(* Logix 5000 project; controller Project_Template vendor 1 type 14 code 106 rev 33.11; software revision 33.00 *)

TASK MainTask (continuous, watchdog 500 ms) : MainProgram

MODULES
   Local : vendor 1 type 14 code 106 (Compact 0, rev 33.11)
      Discrete_In_Slot_3 : 1769-IQ16 (Compact 3, rev 1.1, Input RPI 20 ms)
      Discrete_In_Slot_2 : 1769-IQ16 (Compact 2, rev 1.1, Input RPI 20 ms)
      ASCII_Slot_1 : vendor 1 type 109 code 66 (Compact 1, rev 2.1, Output RPI 2 ms)
      Discrete_Out_Slot_4 : 1769-OW16 (Compact 4, rev 1.1, Output RPI 20 ms)
      Discrete_Out_Slot_5 : 1769-OW16 (Compact 5, rev 1.1, Output RPI 20 ms)
END_MODULES

TYPE BCR_Data :
STRUCT
   LEN : DINT;
   DATA : SINT[9];
END_STRUCT
END_TYPE

TYPE Color_Data :
STRUCT
   LEN : DINT;
   DATA : SINT[4];
END_STRUCT
END_TYPE

VAR_GLOBAL   (* controller tags *)
   I_Auto_Mode_Selector : ALIAS FOR Local:2:I.Data.2;
   I_Barcode_Stop_Raised : ALIAS FOR Local:3:I.Data.1;
   I_Box_Ejector_Extended : ALIAS FOR Local:2:I.Data.4;
   I_Exit_Proxy : ALIAS FOR Local:3:I.Data.7;
   I_Reject_Cyl_Lowered : ALIAS FOR Local:3:I.Data.2;
   I_Reset_PB : ALIAS FOR Local:2:I.Data.3;
   I_Start_PB : ALIAS FOR Local:2:I.Data.0;
   I_Stop_PB : ALIAS FOR Local:2:I.Data.1;
   I_Vacuum_Head_at_Conveyor : ALIAS FOR Local:3:I.Data.0;
   I_Vacuum_Head_at_Magazine : ALIAS FOR Local:2:I.Data.15;
   I_Vacuum_Head_Extended : ALIAS FOR Local:2:I.Data.14;
   I_Vacuum_Head_Lowered : ALIAS FOR Local:2:I.Data.10;
   I_Vacuum_Head_Raised : ALIAS FOR Local:2:I.Data.9;
   I_Vacuum_Head_Retracted : ALIAS FOR Local:2:I.Data.13;
   I_Vacuum_Head_Rotated_CCW : ALIAS FOR Local:2:I.Data.11;
   I_Vacuum_Head_Rotated_CW : ALIAS FOR Local:2:I.Data.12;
   I_Vacuum_Sensor_On : ALIAS FOR Local:3:I.Data.8;
   O_Amber_Tower_Ind : ALIAS FOR Local:5:O.Data.9;
   O_Barcode_Stop_Raise : ALIAS FOR Local:4:O.Data.14;
   O_Box_Eject : ALIAS FOR Local:4:O.Data.0;
   O_Conveyor_On : ALIAS FOR Local:5:O.Data.5;
   O_Green_Tower_Ind : ALIAS FOR Local:5:O.Data.8;
   O_Red_Tower_Ind : ALIAS FOR Local:5:O.Data.10;
   O_Reject_Cyl_Extend : ALIAS FOR Local:5:O.Data.0;
   O_Reject_Cyl_Lower : ALIAS FOR Local:4:O.Data.15;
   O_Vacuum_Head_Extend : ALIAS FOR Local:4:O.Data.8;
   O_Vacuum_Head_Lower : ALIAS FOR Local:4:O.Data.5;
   O_Vacuum_Head_Rotate_CCW : ALIAS FOR Local:4:O.Data.7;
   O_Vacuum_Head_Rotate_CW : ALIAS FOR Local:4:O.Data.6;
   O_Vacuum_Head_to_Conveyor : ALIAS FOR Local:4:O.Data.9;
   O_Vacuum_Head_to_Magazine : ALIAS FOR Local:4:O.Data.10;
   O_Vacuum_Off : ALIAS FOR Local:5:O.Data.2;
   O_Vacuum_On : ALIAS FOR Local:5:O.Data.1;
END_VAR

PROGRAM MainProgram   (* main routine MainRoutine *)
VAR
   barcode_timer : TIMER := (PRE := 3000);
   barcode_timer_1 : TIMER := (PRE := 1500);
   BCR_Good_Read : BOOL;
   BCR_Value : BCR_Data := '33320717$0D';
   Color_Code : DINT := 4;
   Color_Value : Color_Data := '2';
   complete : BOOL;
   Fast_Flash_Off : TIMER := (PRE := 250, ACC := 181, EN := 1, TT := 1);
   Fast_Flash_On : TIMER := (PRE := 250, ACC := 250, EN := 1, DN := 1);
   Fast_Flasher : BOOL := 1;
   Machine_Home : BOOL;
   New_Rx_ID : SINT := 118;
   next_box : BOOL;
   Normal_Flash_Off : TIMER := (PRE := 500);
   Normal_Flash_On : TIMER := (PRE := 500, ACC := 431, EN := 1, TT := 1);
   Old_Rx_ID : SINT := 118;
   Prod_Delay_Timer : TIMER[10] := ([0].PRE := 250, [0].ACC := 250, [0].EN := 1, [0].DN := 1, [1].PRE := 250, [2].PRE := 250, [3].PRE := 250, [4].PRE := 250, [5].PRE := 250, [6].PRE := 250, [7].PRE := 500, [8].PRE := 500);
   Prod_Running : BOOL := 1;
   prod_step : DINT;
   prod_test_bit : DINT := -1;
   Regular_flasher : BOOL;
   Reset_Delay_Timer : TIMER[10] := ([0].PRE := 250, [0].ACC := 250, [0].EN := 1, [0].DN := 1, [1].PRE := 250, [1].ACC := 250, [1].EN := 1, [1].DN := 1, [2].PRE := 250, [2].ACC := 250, [2].EN := 1, [2].DN := 1, [3].PRE := 250, [4].PRE := 250, [4].ACC := 250, [4].EN := 1, [4].DN := 1, [5].PRE := 250, [5].ACC := 250, [5].EN := 1, [5].DN := 1, [6].PRE := 250, [7].PRE := 250);
   Reset_step : DINT := 12;
   Reset_Test_Bit : DINT := -1;
   Resetting : BOOL;
   Slow_Flash_Off : TIMER := (PRE := 1000);
   Slow_Flash_ON : TIMER := (PRE := 1000, ACC := 431, EN := 1, TT := 1);
   Slow_Flasher : BOOL;
   stop_bit : BOOL;
   stop_flag : BOOL := 1;
   stopping : BOOL;
   Test_Bit : DINT;
END_VAR
VAR_INPUT
   dfzsgd : DINT;
END_VAR

ROUTINE a_Reset_Routine   (* ladder *)
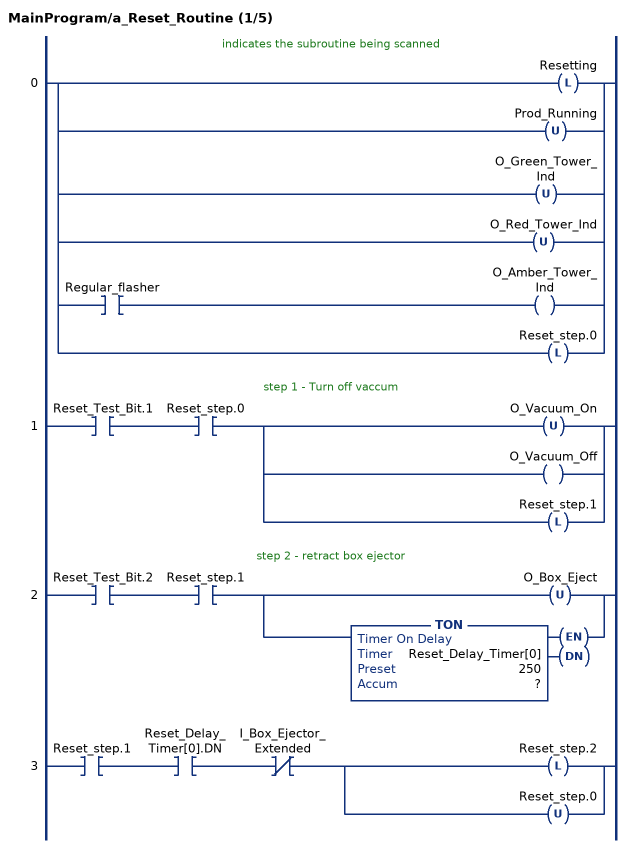
   // indicates the subroutine being scanned
   0: [OTL(Resetting) ,OTU(Prod_Running) ,OTU(O_Green_Tower_Ind) ,OTU(O_Red_Tower_Ind) ,XIC(Regular_flasher) OTE(O_Amber_Tower_Ind) ,OTL(Reset_step.0) ];
   // step 1 - Turn off vaccum
   1: XIC(Reset_Test_Bit.1)XIC(Reset_step.0)[OTU(O_Vacuum_On) ,OTE(O_Vacuum_Off) ,OTL(Reset_step.1) ];
   // step 2 - retract box ejector
   2: XIC(Reset_Test_Bit.2)XIC(Reset_step.1)[OTU(O_Box_Eject) ,TON(Reset_Delay_Timer[0],?,?) ];
   3: XIC(Reset_step.1)XIC(Reset_Delay_Timer[0].DN)XIO(I_Box_Ejector_Extended)[OTL(Reset_step.2) ,OTU(Reset_step.0) ];
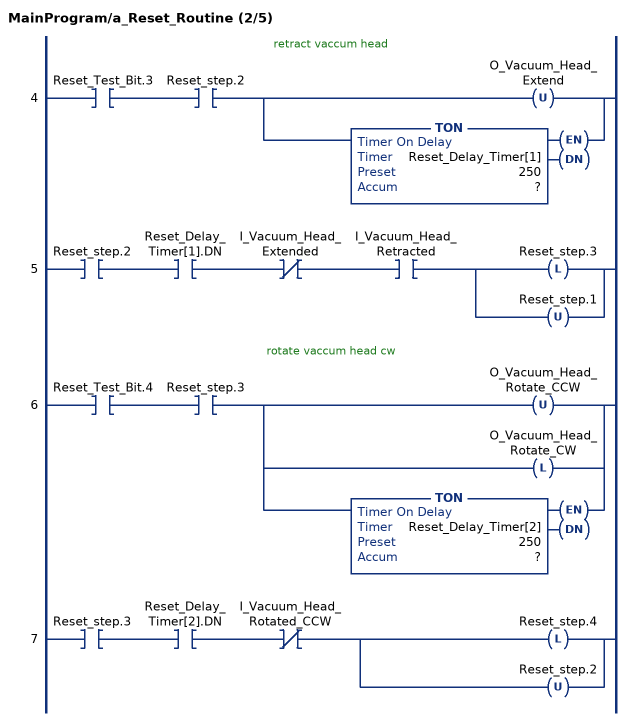
   // retract vaccum head
   4: XIC(Reset_Test_Bit.3)XIC(Reset_step.2)[OTU(O_Vacuum_Head_Extend) ,TON(Reset_Delay_Timer[1],?,?) ];
   5: XIC(Reset_step.2)XIC(Reset_Delay_Timer[1].DN)XIO(I_Vacuum_Head_Extended)XIC(I_Vacuum_Head_Retracted)[OTL(Reset_step.3) ,OTU(Reset_step.1) ];
   // rotate vaccum head cw
   6: XIC(Reset_Test_Bit.4)XIC(Reset_step.3)[OTU(O_Vacuum_Head_Rotate_CCW) ,OTL(O_Vacuum_Head_Rotate_CW) ,TON(Reset_Delay_Timer[2],?,?) ];
   7: XIC(Reset_step.3)XIC(Reset_Delay_Timer[2].DN)XIO(I_Vacuum_Head_Rotated_CCW)[OTL(Reset_step.4) ,OTU(Reset_step.2) ];
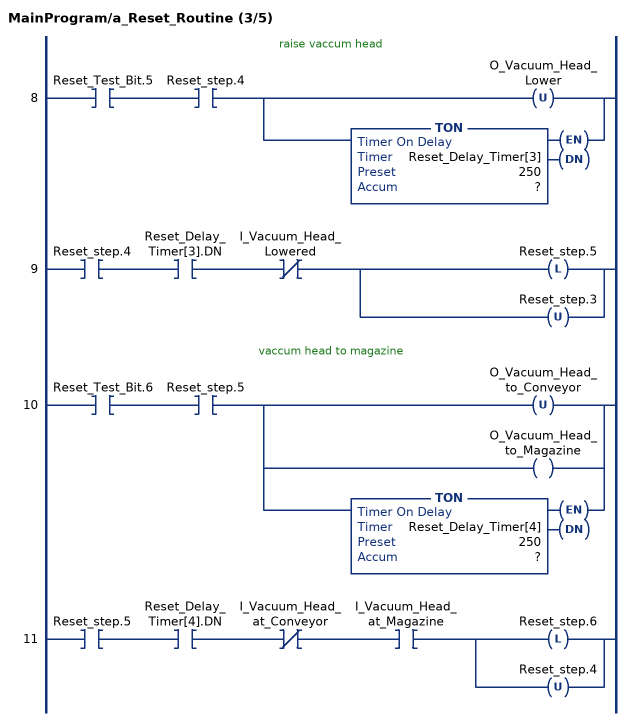
   // raise vaccum head
   8: XIC(Reset_Test_Bit.5)XIC(Reset_step.4)[OTU(O_Vacuum_Head_Lower) ,TON(Reset_Delay_Timer[3],?,?) ];
   9: XIC(Reset_step.4)XIC(Reset_Delay_Timer[3].DN)XIO(I_Vacuum_Head_Lowered)[OTL(Reset_step.5) ,OTU(Reset_step.3) ];
   // vaccum head to magazine
   10: XIC(Reset_Test_Bit.6)XIC(Reset_step.5)[OTU(O_Vacuum_Head_to_Conveyor) ,OTE(O_Vacuum_Head_to_Magazine) ,TON(Reset_Delay_Timer[4],?,?) ];
   11: XIC(Reset_step.5)XIC(Reset_Delay_Timer[4].DN)XIO(I_Vacuum_Head_at_Conveyor)XIC(I_Vacuum_Head_at_Magazine)[OTL(Reset_step.6) ,OTU(Reset_step.4) ];
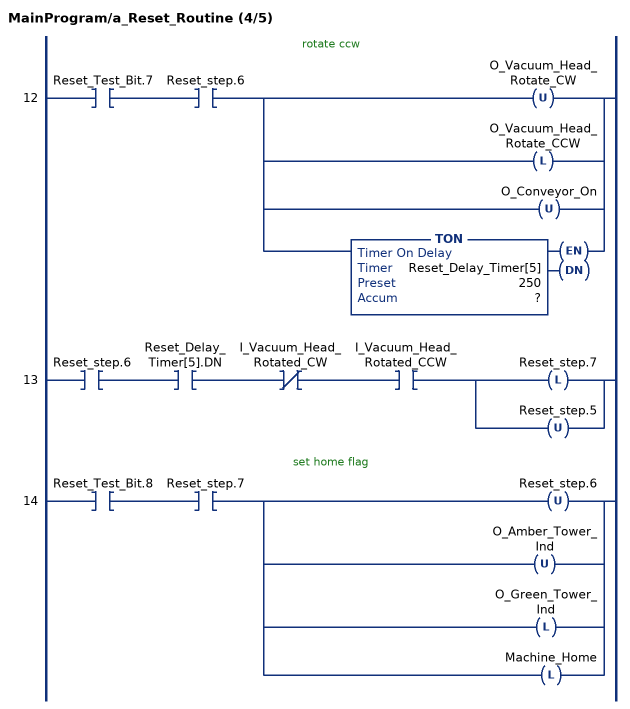
   // rotate ccw
   12: XIC(Reset_Test_Bit.7)XIC(Reset_step.6)[OTU(O_Vacuum_Head_Rotate_CW) ,OTL(O_Vacuum_Head_Rotate_CCW) ,OTU(O_Conveyor_On) ,TON(Reset_Delay_Timer[5],?,?) ];
   13: XIC(Reset_step.6)XIC(Reset_Delay_Timer[5].DN)XIO(I_Vacuum_Head_Rotated_CW)XIC(I_Vacuum_Head_Rotated_CCW)[OTL(Reset_step.7) ,OTU(Reset_step.5) ];
   // set home flag
   14: XIC(Reset_Test_Bit.8)XIC(Reset_step.7)[OTU(Reset_step.6) ,OTU(O_Amber_Tower_Ind) ,OTL(O_Green_Tower_Ind) ,OTL(Machine_Home) ];
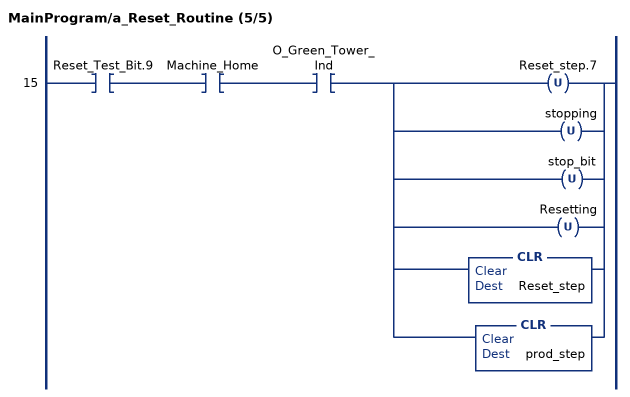
   15: XIC(Reset_Test_Bit.9)XIC(Machine_Home)XIC(O_Green_Tower_Ind)[OTU(Reset_step.7) ,OTU(stopping) ,OTU(stop_bit) ,OTU(Resetting) ,CLR(Reset_step) ,CLR(prod_step) ];
END_ROUTINE

ROUTINE Auto_Routine   (* ladder *)
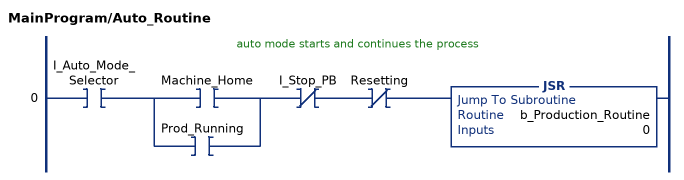
   // auto mode starts and continues the process
   0: XIC(I_Auto_Mode_Selector)[XIC(Machine_Home) ,XIC(Prod_Running) ]XIO(I_Stop_PB)XIO(Resetting)JSR(b_Production_Routine,0);
END_ROUTINE

ROUTINE b_Production_Routine   (* ladder *)
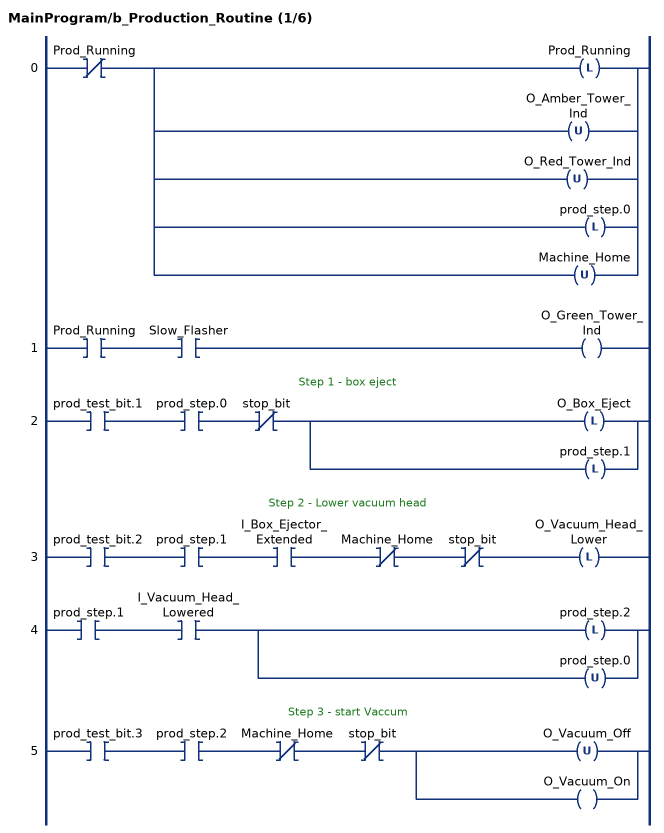
   0: XIO(Prod_Running)[OTL(Prod_Running) ,OTU(O_Amber_Tower_Ind) ,OTU(O_Red_Tower_Ind) ,OTL(prod_step.0) ,OTU(Machine_Home) ];
   1: XIC(Prod_Running)XIC(Slow_Flasher)OTE(O_Green_Tower_Ind);
   // Step 1 - box eject
   2: XIC(prod_test_bit.1)XIC(prod_step.0)XIO(stop_bit)[OTL(O_Box_Eject) ,OTL(prod_step.1) ];
   // Step 2 - Lower vacuum head
   3: XIC(prod_test_bit.2)XIC(prod_step.1)XIC(I_Box_Ejector_Extended)XIO(Machine_Home)XIO(stop_bit)OTL(O_Vacuum_Head_Lower);
   4: XIC(prod_step.1)XIC(I_Vacuum_Head_Lowered)[OTL(prod_step.2) ,OTU(prod_step.0) ];
   // Step 3 - start Vaccum
   5: XIC(prod_test_bit.3)XIC(prod_step.2)XIO(Machine_Home)XIO(stop_bit)[OTU(O_Vacuum_Off) ,OTE(O_Vacuum_On) ];
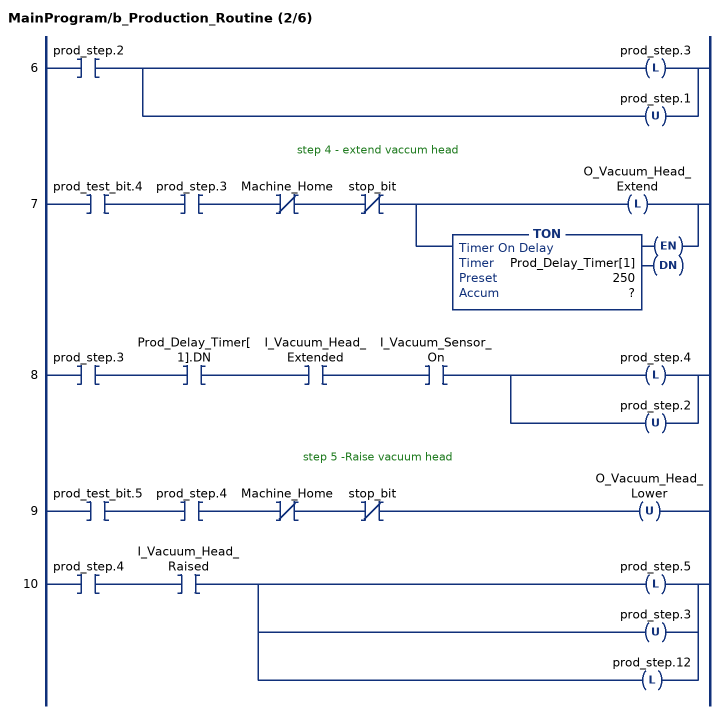
   6: XIC(prod_step.2)[OTL(prod_step.3) ,OTU(prod_step.1) ];
   // step 4 - extend vaccum head
   7: XIC(prod_test_bit.4)XIC(prod_step.3)XIO(Machine_Home)XIO(stop_bit)[OTL(O_Vacuum_Head_Extend) ,TON(Prod_Delay_Timer[1],?,?) ];
   8: XIC(prod_step.3)XIC(Prod_Delay_Timer[1].DN)XIC(I_Vacuum_Head_Extended)XIC(I_Vacuum_Sensor_On)[OTL(prod_step.4) ,OTU(prod_step.2) ];
   // step 5 -Raise vacuum head
   9: XIC(prod_test_bit.5)XIC(prod_step.4)XIO(Machine_Home)XIO(stop_bit)OTU(O_Vacuum_Head_Lower);
   10: XIC(prod_step.4)XIC(I_Vacuum_Head_Raised)[OTL(prod_step.5) ,OTU(prod_step.3) ,OTL(prod_step.12) ];
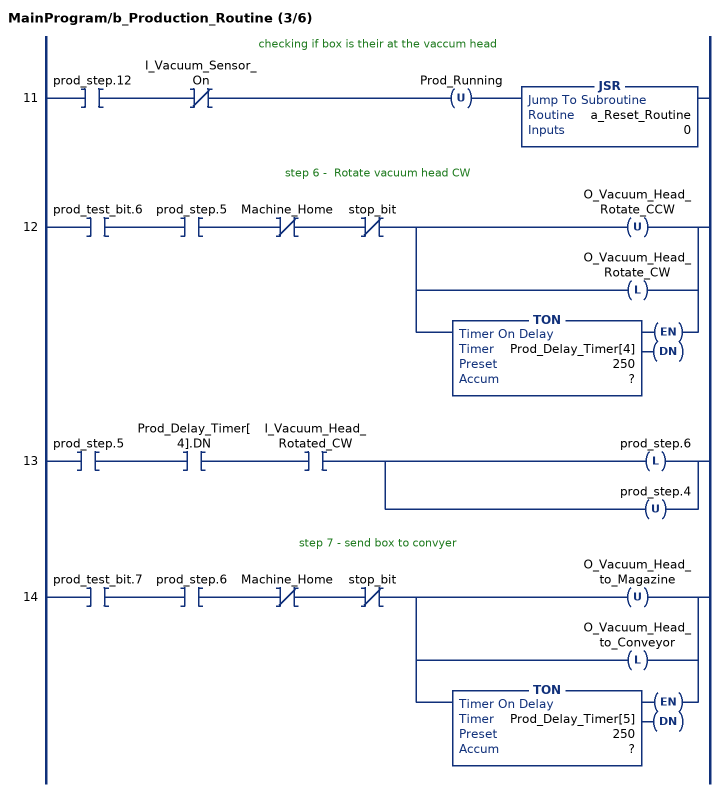
   // checking if box is their at the vaccum head
   11: XIC(prod_step.12)XIO(I_Vacuum_Sensor_On)OTU(Prod_Running)JSR(a_Reset_Routine,0);
   // step 6 -  Rotate vacuum head CW
   12: XIC(prod_test_bit.6)XIC(prod_step.5)XIO(Machine_Home)XIO(stop_bit)[OTU(O_Vacuum_Head_Rotate_CCW) ,OTL(O_Vacuum_Head_Rotate_CW) ,TON(Prod_Delay_Timer[4],?,?) ];
   13: XIC(prod_step.5)XIC(Prod_Delay_Timer[4].DN)XIC(I_Vacuum_Head_Rotated_CW)[OTL(prod_step.6) ,OTU(prod_step.4) ];
   // step 7 - send box to convyer
   14: XIC(prod_test_bit.7)XIC(prod_step.6)XIO(Machine_Home)XIO(stop_bit)[OTU(O_Vacuum_Head_to_Magazine) ,OTL(O_Vacuum_Head_to_Conveyor) ,TON(Prod_Delay_Timer[5],?,?) ];
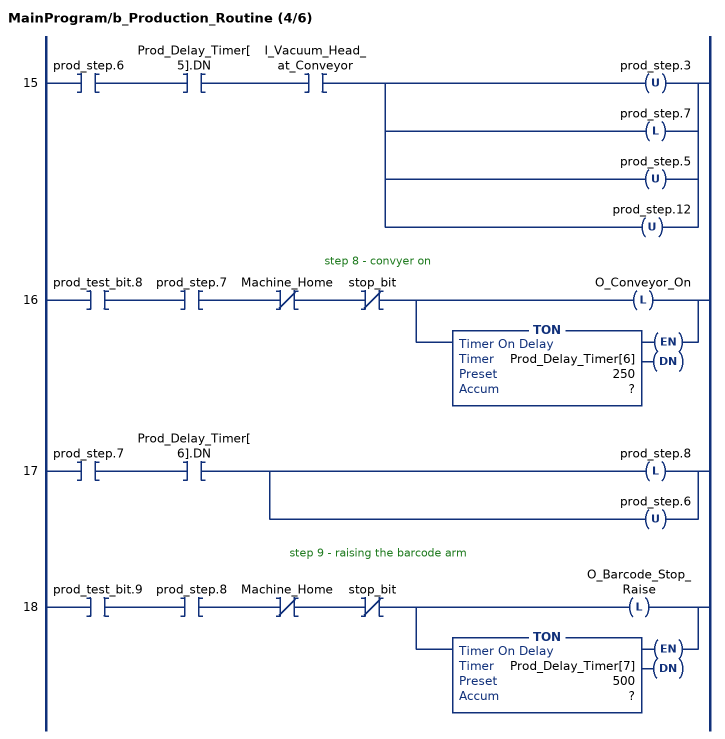
   15: XIC(prod_step.6)XIC(Prod_Delay_Timer[5].DN)XIC(I_Vacuum_Head_at_Conveyor)[OTU(prod_step.3) ,OTL(prod_step.7) ,OTU(prod_step.5) ,OTU(prod_step.12) ];
   // step 8 - convyer on
   16: XIC(prod_test_bit.8)XIC(prod_step.7)XIO(Machine_Home)XIO(stop_bit)[OTL(O_Conveyor_On) ,TON(Prod_Delay_Timer[6],?,?) ];
   17: XIC(prod_step.7)XIC(Prod_Delay_Timer[6].DN)[OTL(prod_step.8) ,OTU(prod_step.6) ];
   // step 9 - raising the barcode arm
   18: XIC(prod_test_bit.9)XIC(prod_step.8)XIO(Machine_Home)XIO(stop_bit)[OTL(O_Barcode_Stop_Raise) ,TON(Prod_Delay_Timer[7],?,?) ];
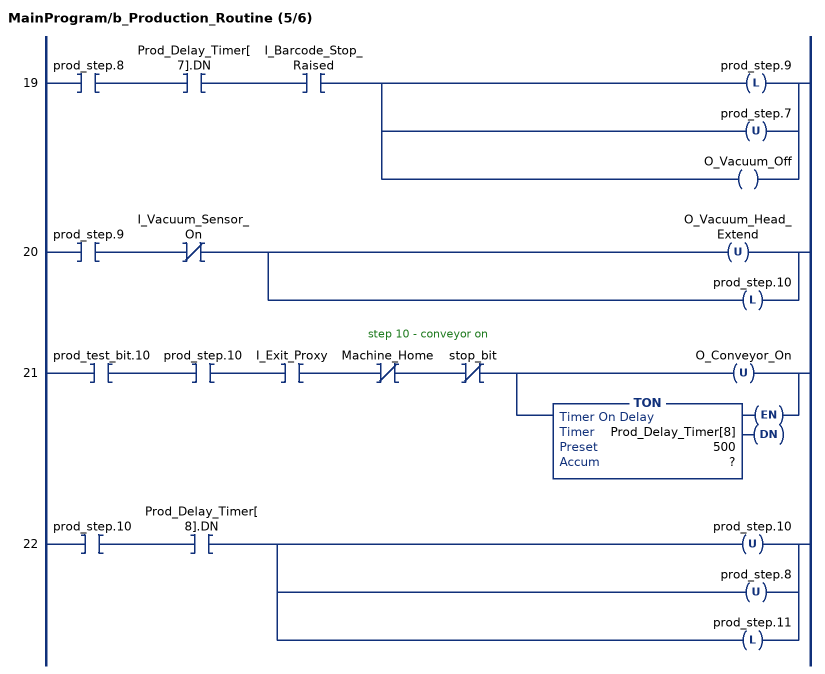
   19: XIC(prod_step.8)XIC(Prod_Delay_Timer[7].DN)XIC(I_Barcode_Stop_Raised)[OTL(prod_step.9) ,OTU(prod_step.7) ,OTE(O_Vacuum_Off) ];
   20: XIC(prod_step.9)XIO(I_Vacuum_Sensor_On)[OTU(O_Vacuum_Head_Extend) ,OTL(prod_step.10) ];
   // step 10 - conveyor on
   21: XIC(prod_test_bit.10)XIC(prod_step.10)XIC(I_Exit_Proxy)XIO(Machine_Home)XIO(stop_bit)[OTU(O_Conveyor_On) ,TON(Prod_Delay_Timer[8],?,?) ];
   22: XIC(prod_step.10)XIC(Prod_Delay_Timer[8].DN)[OTU(prod_step.10) ,OTU(prod_step.8) ,OTL(prod_step.11) ];
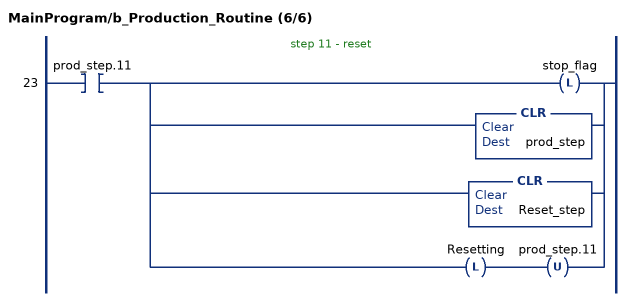
   // step 11 - reset
   23: XIC(prod_step.11)[OTL(stop_flag) ,CLR(prod_step) ,CLR(Reset_step) ,OTL(Resetting) OTU(prod_step.11) ];
END_ROUTINE

ROUTINE barcode_scan_routine   (* ladder *)
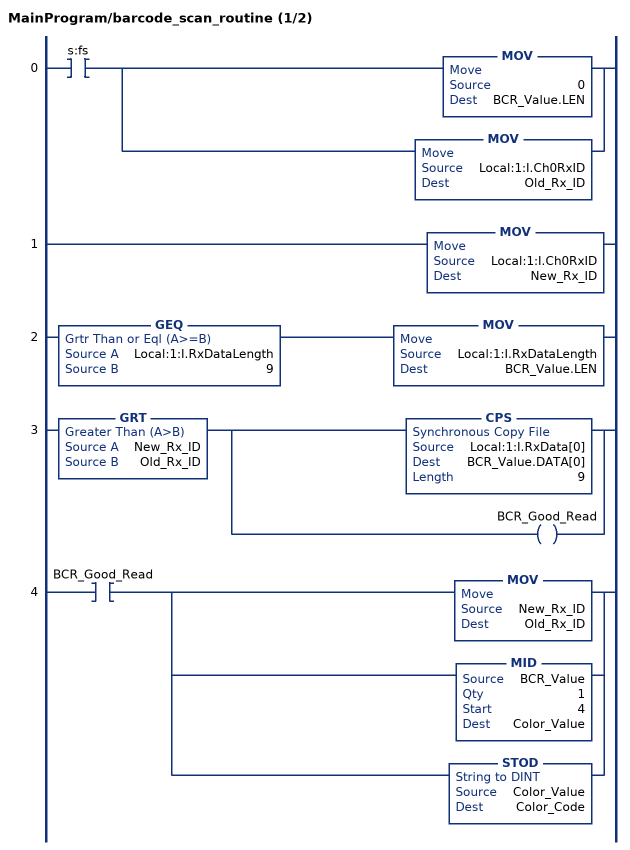
   0: XIC(s:fs)[MOV(0,BCR_Value.LEN) ,MOV(Local:1:I.Ch0RxID,Old_Rx_ID) ];
   1: MOV(Local:1:I.Ch0RxID,New_Rx_ID);
   2: GEQ(Local:1:I.RxDataLength,9)MOV(Local:1:I.RxDataLength,BCR_Value.LEN);
   3: GRT(New_Rx_ID,Old_Rx_ID)[CPS(Local:1:I.RxData[0],BCR_Value.DATA[0],9) ,OTE(BCR_Good_Read) ];
   4: XIC(BCR_Good_Read)[MOV(New_Rx_ID,Old_Rx_ID) ,MID(BCR_Value,1,4,Color_Value) ,STOD(Color_Value,Color_Code) ];
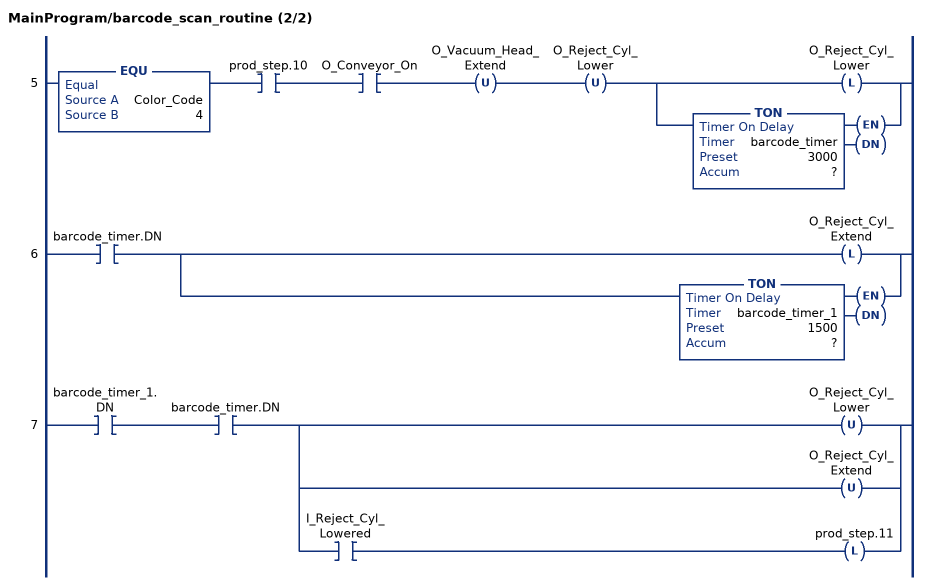
   5: EQU(Color_Code,4)XIC(prod_step.10)XIC(O_Conveyor_On)OTU(O_Vacuum_Head_Extend)OTU(O_Reject_Cyl_Lower)[OTL(O_Reject_Cyl_Lower) ,TON(barcode_timer,?,?) ];
   6: XIC(barcode_timer.DN)[OTL(O_Reject_Cyl_Extend) ,TON(barcode_timer_1,?,?) ];
   7: XIC(barcode_timer_1.DN)XIC(barcode_timer.DN)[OTU(O_Reject_Cyl_Lower) ,OTU(O_Reject_Cyl_Extend) ,XIC(I_Reject_Cyl_Lowered) OTL(prod_step.11) ];
END_ROUTINE

ROUTINE MainRoutine   (* ladder *)
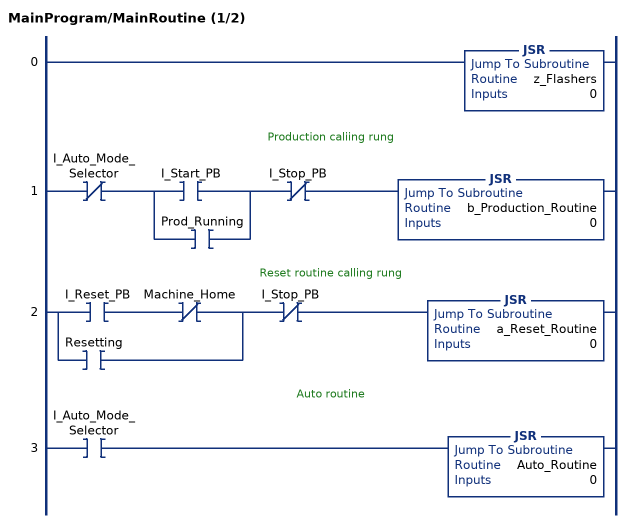
   0: JSR(z_Flashers,0);
   // Production caliing rung
   1: XIO(I_Auto_Mode_Selector)[XIC(I_Start_PB) ,XIC(Prod_Running) ]XIO(I_Stop_PB)JSR(b_Production_Routine,0);
   // Reset routine calling rung
   2: [XIC(I_Reset_PB) XIO(Machine_Home) ,XIC(Resetting) ]XIO(I_Stop_PB)JSR(a_Reset_Routine,0);
   // Auto routine
   3: XIC(I_Auto_Mode_Selector)JSR(Auto_Routine,0);
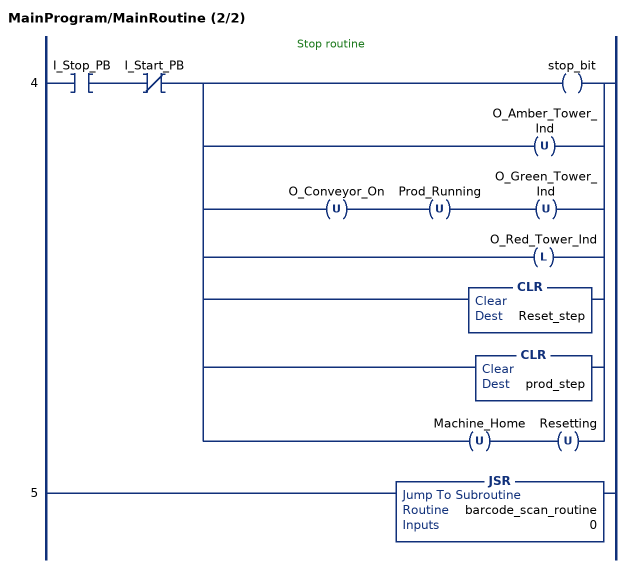
   // Stop routine
   4: XIC(I_Stop_PB)XIO(I_Start_PB)[OTE(stop_bit) ,OTU(O_Amber_Tower_Ind) ,OTU(O_Conveyor_On) OTU(Prod_Running) OTU(O_Green_Tower_Ind) ,OTL(O_Red_Tower_Ind) ,CLR(Reset_step) ,CLR(prod_step) ,OTU(Machine_Home) OTU(Resetting) ];
   5: JSR(barcode_scan_routine,0);
END_ROUTINE

ROUTINE z_Flashers   (* ladder *)
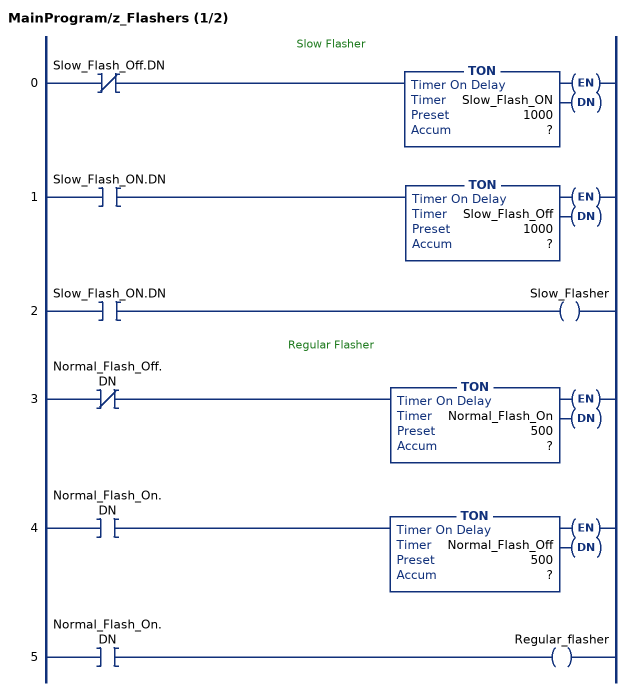
   // Slow Flasher
   0: XIO(Slow_Flash_Off.DN)TON(Slow_Flash_ON,?,?);
   1: XIC(Slow_Flash_ON.DN)TON(Slow_Flash_Off,?,?);
   2: XIC(Slow_Flash_ON.DN)OTE(Slow_Flasher);
   // Regular Flasher
   3: XIO(Normal_Flash_Off.DN)TON(Normal_Flash_On,?,?);
   4: XIC(Normal_Flash_On.DN)TON(Normal_Flash_Off,?,?);
   5: XIC(Normal_Flash_On.DN)OTE(Regular_flasher);
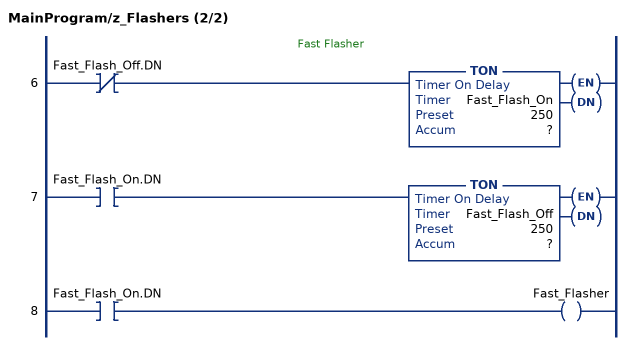
   // Fast Flasher
   6: XIO(Fast_Flash_Off.DN)TON(Fast_Flash_On,?,?);
   7: XIC(Fast_Flash_On.DN)TON(Fast_Flash_Off,?,?);
   8: XIC(Fast_Flash_On.DN)OTE(Fast_Flasher);
END_ROUTINE
END_PROGRAM
